FUNCTION_BLOCK CAN_Example
VAR_INPUT
END_VAR
VAR_OUTPUT
END_VAR
VAR
	fPhase1_Uptime	: DINT;
	fPhase2_Uptime	: DINT;
	fPhase3_Uptime	: DINT;
	fPhase1_Offset	: DINT;
	fPhase2_Offset	: DINT;
	fPhase3_Offset	: DINT;
END_VAR

(*
Example codes from some beckhoff PDF

Sample code: Sending messages from the PLC
if Outputs.TxCounter = Inputs.TxCounter then
          for i=0 to NumberOfMessagesToSend do
                  Outputs.TxMessage[i] = MessageToSend[i];
          End_for
          Outputs.NoOfTxMessages = NumberOfMessagesToSend;
          Outputs.TxCounter := Outputs.TxCounter + 1;
end_if


Sample code: Receiving messages from the PLC
if Outputs.RxCounter <> Inputs.RxCounter then
          for I := 0 to (Inputs.NoOfRxMessages-1) do
                   MessageReceived[i] := Inputs.RxMessage [i];
          End_for
          Outputs.RxCounter := Outputs.RxCounter+1;
end_if

*)

END_FUNCTION_BLOCK

(* stored: Version 1.1.0.1, ProductVersion 3.1.4022.17
   POU CAN_Example: Id {1daa8427-a4bf-4d32-a0f1-8e66064ac444}, SpecialFunc None *)
